(* CODESYS project sensata_io.library
   Company: Sensata Technologies
   DocFormat: reStructuredText
   Description: Contains IO structs for easy linking to IO
   Version: 0.0.1
   Placeholder: Sensata_IO
   Title: Sensata_IO

Project tree, tasks and I/O mapping:
  libraries: Tc2_Standard, * (Beckhoff Automation GmbH); Tc2_System, * (Beckhoff Automation GmbH); Tc2_Utilities, * (Beckhoff Automation GmbH); Tc3_Module, * (Beckhoff Automation GmbH)
  Beckhoff/
    EL1xxx/
      data type ST_EL1008
      data type ST_EL1008_Inputs
      data type ST_EL1014
      data type ST_EL1014_Inputs
      data type ST_EL1258
      data type ST_EL1258_Inputs
      data type ST_EL1258_Inputs_Channel
      data type ST_EL1258_Inputs_Channel_EventStates
      data type ST_EL1258_Inputs_Channel_Status
      data type ST_EL1258_Outputs
      data type ST_EL1258_Outputs_Channel
    EL2xxx/
      data type ST_EL2004
      data type ST_EL2004_Outputs
      data type ST_EL2008
      data type ST_EL2008_Outputs
      data type ST_EL2624
      data type ST_EL2624_Outputs
    EL3xxx/
      data type ST_EL3104
      data type ST_EL3104_Inputs
      data type ST_EL3104_Inputs_Channel
      data type ST_EL3104_Inputs_Channel_Status
      data type ST_EL3704_24BitVoltageDiff
      data type ST_EL3704_24BitVoltageDiff_Inputs
      data type ST_EL3704_24BitVoltageDiff_Inputs_Status
      data type ST_EL3773
      data type ST_EL3773_Inputs
      data type ST_EL3773_Inputs_Channel
      data type ST_EL3773_Inputs_Channel_Status
    EP1xxx/
      data type ST_EP1008
      data type ST_EP1008_Inputs
  IO Debug/
    function F_LinkDigitalIOStructs [ST]
    function F_SetDigitalInput [ST]
    function F_SetDigitalOutput [ST]
    data type ST_DebugDigitalIO
  Keyence/
    Barcode Scanners/
      data type ST_KeyenceNL20_EIP
      data type ST_KeyenceNL20_EIP_Inputs
      data type ST_KeyenceNL20_EIP_Outputs
      data type ST_KeyenceSR750_EIP
      data type ST_KeyenceSR750_EIP_Inputs
      data type ST_KeyenceSR750_EIP_Outputs
      data type ST_KeyenceSRX1H3H_EIP
      data type ST_KeyenceSRX1H3H_EIP_Inputs
      data type ST_KeyenceSRX1H3H_EIP_Outputs
    Height Check/
      data type ST_DLEC1A
      data type ST_DLEC1A_Inputs
      data type ST_DLEC1A_Inputs_Response
      data type ST_DLEC1A_Inputs_SystemStatus
      data type ST_DLEC1A_Outputs
      data type ST_DLEC1A_Outputs_Request
    Safety PLCs/
    Sensors/
      data type ST_LRX100
      data type ST_LRX100_Inputs
      data type ST_LRX100_Outputs
  MurrElektronik/
    data type ST_IMPACT67
    data type ST_IMPACT67_Inputs
  Norgren/
    data type ST_VR10
    data type ST_VR10_Inputs
    data type ST_VR10_Outputs
  SMC/
    data type ST_SMCEX260SEC3
    data type ST_SMCEX260SEC3_32Bit
    data type ST_SMCEX260SEC3_32Bit_Outputs
    data type ST_SMCEX260SEC3_Outputs
*)

// Beckhoff/EL1xxx/ST_EL1008
TYPE ST_EL1008 :
STRUCT
	stIn AT %I*: ST_EL1008_Inputs;
END_STRUCT
END_TYPE

// Beckhoff/EL1xxx/ST_EL1008_Inputs
TYPE ST_EL1008_Inputs :
STRUCT
	bitInput1: BIT;
	bitInput2: BIT;
	bitInput3: BIT;
	bitInput4: BIT;
	bitInput5: BIT;
	bitInput6: BIT;
	bitInput7: BIT;
	bitInput8: BIT;
END_STRUCT
END_TYPE

// Beckhoff/EL1xxx/ST_EL1014
TYPE ST_EL1014 :
STRUCT
	stIn AT %I*: ST_EL1014_Inputs;
END_STRUCT
END_TYPE

// Beckhoff/EL1xxx/ST_EL1014_Inputs
TYPE ST_EL1014_Inputs :
STRUCT
	bitInput1: BIT;
	bitInput2: BIT;
	bitInput3: BIT;
	bitInput4: BIT;
END_STRUCT
END_TYPE

// Beckhoff/EL1xxx/ST_EL1258
TYPE ST_EL1258 :
STRUCT
	stIn AT %I*: ST_EL1258_Inputs;
	stOut AT %Q*: ST_EL1258_Outputs;
END_STRUCT
END_TYPE

// Beckhoff/EL1xxx/ST_EL1258_Inputs
TYPE ST_EL1258_Inputs :
STRUCT
	stChannel1: ST_EL1258_Inputs_Channel;
	stChannel2: ST_EL1258_Inputs_Channel;
	stChannel3: ST_EL1258_Inputs_Channel;
	stChannel4: ST_EL1258_Inputs_Channel;
	stChannel5: ST_EL1258_Inputs_Channel;
	stChannel6: ST_EL1258_Inputs_Channel;
	stChannel7: ST_EL1258_Inputs_Channel;
	stChannel8: ST_EL1258_Inputs_Channel;
END_STRUCT
END_TYPE

// Beckhoff/EL1xxx/ST_EL1258_Inputs_Channel
TYPE ST_EL1258_Inputs_Channel :
STRUCT
	stStatus: ST_EL1258_Inputs_Channel_Status;
	stEventStates: ST_EL1258_Inputs_Channel_EventStates;
	arrEventTime: ARRAY[1..10] OF UDINT;
END_STRUCT
END_TYPE

// Beckhoff/EL1xxx/ST_EL1258_Inputs_Channel_EventStates
TYPE ST_EL1258_Inputs_Channel_EventStates :
STRUCT
	bitEventState01: BIT;
	bitEventState02: BIT;
	bitEventState03: BIT;
	bitEventState04: BIT;
	bitEventState05: BIT;
	bitEventState06: BIT;
	bitEventState07: BIT;
	bitEventState08: BIT;
	bitEventState09: BIT;
	bitEventState10: BIT;
END_STRUCT
END_TYPE

// Beckhoff/EL1xxx/ST_EL1258_Inputs_Channel_Status
TYPE ST_EL1258_Inputs_Channel_Status :
STRUCT
	usintEventsCount: USINT;
	
	bitState: BIT;
	bitBufferOverflow: BIT;
	{attribute 'hide'}
	bitReserved022: BIT;
	{attribute 'hide'}
	bitReserved023: BIT;
	{attribute 'hide'}
	bitReserved024: BIT;
	{attribute 'hide'}
	bitReserved25: BIT;
	bitCycleCountBit0: BIT;
	bitCycleCountBit1: BIT;
	
	usintBufferEvents: USINT;
	usintOrderFeedback: USINT;
END_STRUCT
END_TYPE

// Beckhoff/EL1xxx/ST_EL1258_Outputs
TYPE ST_EL1258_Outputs :
STRUCT
	stChannel1: ST_EL1258_Outputs_Channel;
	stChannel2: ST_EL1258_Outputs_Channel;
	stChannel3: ST_EL1258_Outputs_Channel;
	stChannel4: ST_EL1258_Outputs_Channel;
	stChannel5: ST_EL1258_Outputs_Channel;
	stChannel6: ST_EL1258_Outputs_Channel;
	stChannel7: ST_EL1258_Outputs_Channel;
	stChannel8: ST_EL1258_Outputs_Channel;
END_STRUCT
END_TYPE

// Beckhoff/EL1xxx/ST_EL1258_Outputs_Channel
TYPE ST_EL1258_Outputs_Channel :
STRUCT
	bitBufferReset: BIT;
	{attribute 'hide'}
	bitReserved01: BIT;
	{attribute 'hide'}
	bitReserved02: BIT;
	{attribute 'hide'}
	bitReserved03: BIT;
	{attribute 'hide'}
	bitReserved04: BIT;
	{attribute 'hide'}
	bitReserved05: BIT;
	{attribute 'hide'}
	bitReserved06: BIT;
	{attribute 'hide'}
	bitReserved07: BIT;
	
	{attribute 'hide'}
	byteReserved10: BYTE;
	
	usintInputOrderCounter: BOOL;
END_STRUCT
END_TYPE

// Beckhoff/EL2xxx/ST_EL2004
TYPE ST_EL2004 :
STRUCT
	stOut AT %Q*: ST_EL2004_Outputs;
END_STRUCT
END_TYPE

// Beckhoff/EL2xxx/ST_EL2004_Outputs
TYPE ST_EL2004_Outputs :
STRUCT
	bitOutput1: BIT;
	bitOutput2: BIT;
	bitOutput3: BIT;
	bitOutput4: BIT;
END_STRUCT
END_TYPE

// Beckhoff/EL2xxx/ST_EL2008
TYPE ST_EL2008 :
STRUCT
	stOut AT %Q*: ST_EL2008_Outputs;
END_STRUCT
END_TYPE

// Beckhoff/EL2xxx/ST_EL2008_Outputs
TYPE ST_EL2008_Outputs :
STRUCT
	bitOutput1: BIT;
	bitOutput2: BIT;
	bitOutput3: BIT;
	bitOutput4: BIT;
	bitOutput5: BIT;
	bitOutput6: BIT;
	bitOutput7: BIT;
	bitOutput8: BIT;
END_STRUCT
END_TYPE

// Beckhoff/EL2xxx/ST_EL2624
TYPE ST_EL2624 :
STRUCT
	stOut AT %Q*: ST_EL2624_Outputs;
END_STRUCT
END_TYPE

// Beckhoff/EL2xxx/ST_EL2624_Outputs
TYPE ST_EL2624_Outputs :
STRUCT
	bitRelay1: BIT;
	bitRelay2: BIT;
	bitRelay3: BIT;
	bitRelay4: BIT;
END_STRUCT
END_TYPE

// Beckhoff/EL3xxx/ST_EL3104
TYPE ST_EL3104 :
STRUCT
	stIn AT %I*: ST_EL3104_Inputs;
END_STRUCT
END_TYPE

// Beckhoff/EL3xxx/ST_EL3104_Inputs
TYPE ST_EL3104_Inputs :
STRUCT
	stChannel1: ST_EL3104_Inputs_Channel;
	stChannel2: ST_EL3104_Inputs_Channel;
	stChannel3: ST_EL3104_Inputs_Channel;
	stChannel4: ST_EL3104_Inputs_Channel;
END_STRUCT
END_TYPE

// Beckhoff/EL3xxx/ST_EL3104_Inputs_Channel
TYPE ST_EL3104_Inputs_Channel :
STRUCT
	stStatus: ST_EL3104_Inputs_Channel_Status;
	intValue: INT;
END_STRUCT
END_TYPE

// Beckhoff/EL3xxx/ST_EL3104_Inputs_Channel_Status
TYPE ST_EL3104_Inputs_Channel_Status :
STRUCT
	bitUnderRange: BIT;
	bitOverRange: BIT;
	bitOverLimit1: BIT;
	bitUnderLimit1: BIT;
	bitOverLimit2: BIT;
	bitUnderLimit2: BIT;
	bitError: BIT;
	{attribute 'hide'}
	bitReserved07: BIT;
	
	{attribute 'hide'}
	bitReserved10: BIT;
	{attribute 'hide'}
	bitReserved11: BIT;
	{attribute 'hide'}
	bitReserved12: BIT;
	{attribute 'hide'}
	bitReserved13: BIT;
	{attribute 'hide'}
	bitReserved14: BIT;
	bitSyncError: BIT;
	bitTxPDOState: BIT;
	bitTxPDOToggle: BIT;
END_STRUCT
END_TYPE

// Beckhoff/EL3xxx/ST_EL3704_24BitVoltageDiff
TYPE ST_EL3704_24BitVoltageDiff :
STRUCT
	stIn AT %I*: ST_EL3704_24BitVoltageDiff_Inputs;
END_STRUCT
END_TYPE

// Beckhoff/EL3xxx/ST_EL3704_24BitVoltageDiff_Inputs
TYPE ST_EL3704_24BitVoltageDiff_Inputs :
STRUCT
	stChannel1Status: ST_EL3704_24BitVoltageDiff_Inputs_Status;
	dintChannel1Value: DINT;
	ulintChannel1Timestamp: ULINT;
	stChannel2Status: ST_EL3704_24BitVoltageDiff_Inputs_Status;
	dintChannel2Value: DINT;
	stChannel3Status: ST_EL3704_24BitVoltageDiff_Inputs_Status;
	dintChannel3Value: DINT;
	stChannel4Status: ST_EL3704_24BitVoltageDiff_Inputs_Status;
	dintChannel4Value: DINT;
END_STRUCT
END_TYPE

// Beckhoff/EL3xxx/ST_EL3704_24BitVoltageDiff_Inputs_Status
TYPE ST_EL3704_24BitVoltageDiff_Inputs_Status :
STRUCT
	usintSamples: USINT;
	bitError: BIT;
	bitUnderrange: BIT;
	bitOverrange: BIT;
	{attribute 'hide'}
	bitReserved13: BIT;
	bitDiag: BIT;
	bitTxPDOState: BIT;
	bitCycleCount1: BIT;
	bitCycleCount2: BIT;
END_STRUCT
END_TYPE

// Beckhoff/EL3xxx/ST_EL3773
TYPE ST_EL3773 :
STRUCT
	stIn AT %I*: ST_EL3773_Inputs;
END_STRUCT
END_TYPE

// Beckhoff/EL3xxx/ST_EL3773_Inputs
TYPE ST_EL3773_Inputs :
STRUCT
	stL1: ST_EL3773_Inputs_Channel;
	stL2: ST_EL3773_Inputs_Channel;
	stL3: ST_EL3773_Inputs_Channel;
	udintNextSyncTimeLow: UDINT;
	udintNextSyncTimeHigh: UDINT;
	uintSampleCount: UINT;
END_STRUCT
END_TYPE

// Beckhoff/EL3xxx/ST_EL3773_Inputs_Channel
TYPE ST_EL3773_Inputs_Channel :
STRUCT
	stVoltageStatus: ST_EL3773_Inputs_Channel_Status;
	arrVoltageSamples: ARRAY[0..9] OF INT;
	stCurrentStatus: ST_EL3773_Inputs_Channel_Status;
	arrCurrentSamples: ARRAY[0..9] OF INT;
END_STRUCT
END_TYPE

// Beckhoff/EL3xxx/ST_EL3773_Inputs_Channel_Status
TYPE ST_EL3773_Inputs_Channel_Status :
STRUCT
	bitUnderRange: BIT;
	bitOverRange: BIT;
	bitOverLimit: BIT;
	bitUnderLimit: BIT;
	{attribute 'hide'}
	bitReserved04: BIT;
	{attribute 'hide'}
	bitReserved05: BIT;
	bitError: BIT;
	{attribute 'hide'}
	bitReserved07: BIT;
	
	{attribute 'hide'}
	bitReserved10: BIT;
	{attribute 'hide'}
	bitReserved11: BIT;
	{attribute 'hide'}
	bitReserved12: BIT;
	{attribute 'hide'}
	bitReserved13: BIT;
	{attribute 'hide'}
	bitReserved14: BIT;
	bitSyncError: BIT;
	bitTxPDOState: BIT;
	bitTxPDOToggle: BIT;
END_STRUCT
END_TYPE

// Beckhoff/EP1xxx/ST_EP1008
TYPE ST_EP1008 :
STRUCT
	stIn AT %I*: ST_EP1008_Inputs;
END_STRUCT
END_TYPE

// Beckhoff/EP1xxx/ST_EP1008_Inputs
TYPE ST_EP1008_Inputs :
STRUCT
	bitInput1: BIT;
	bitInput2: BIT;
	bitInput3: BIT;
	bitInput4: BIT;
	bitInput5: BIT;
	bitInput6: BIT;
	bitInput7: BIT;
	bitInput8: BIT;
END_STRUCT
END_TYPE

// IO Debug/ST_DebugDigitalIO
TYPE ST_DebugDigitalIO :
STRUCT
	(* Label for this IO. *)
	strLabel: T_MaxString;
	(* Current value. *)
	bCurrentValue: BOOL;
	(* Set to TRUE if IO is an output. *)
	bOutput: BOOL;
	(* Set TRUE to force output to a value. *)
	bForce: BOOL;
	(* Value to force output to. *)
	bForceValue: BOOL;
END_STRUCT
END_TYPE

// Keyence/Barcode Scanners/ST_KeyenceNL20_EIP
TYPE ST_KeyenceNL20_EIP :
STRUCT
	stIn AT %I*: ST_KeyenceNL20_EIP_Inputs;
	stOut AT %Q*: ST_KeyenceNL20_EIP_Outputs;
END_STRUCT
END_TYPE

// Keyence/Barcode Scanners/ST_KeyenceNL20_EIP_Inputs
TYPE ST_KeyenceNL20_EIP_Inputs :
STRUCT
	bitError: BIT;
	bitResponseDataAvailable: BIT;
	bitResultDataStrobe: BIT;
	{attribute 'hide'}
	bitReserved003: BIT;
	{attribute 'hide'}
	bitReserved004: BIT;
	{attribute 'hide'}
	bitReserved005: BIT;
	bitBufferOverflowError: BIT;
	bitGeneralError: BIT;
	
	bitBusy: BIT;
	{attribute 'hide'}
	bitReserved011: BIT;
	{attribute 'hide'}
	bitReserved012: BIT;
	bitModeBusy: BIT;
	{attribute 'hide'}
	bitReserved014: BIT;
	{attribute 'hide'}
	bitReserved015: BIT;
	{attribute 'hide'}
	bitReserved016: BIT;
	{attribute 'hide'}
	bitReserved017: BIT;
	
	bitReadComplete: BIT;
	{attribute 'hide'}
	bitReserved021: BIT;
	{attribute 'hide'}
	bitReserved022: BIT;
	{attribute 'hide'}
	bitReserved023: BIT;
	{attribute 'hide'}
	bitReserved024: BIT;
	{attribute 'hide'}
	bitReserved025: BIT;
	{attribute 'hide'}
	bitReserved026: BIT;
	{attribute 'hide'}
	bitReserved027: BIT;
	
	{attribute 'hide'}
	byteReserved030: BYTE;

	bitIN1Status: BIT;
	bitIN2Status: BIT;
	{attribute 'hide'}
	bitReserved042: BIT;
	{attribute 'hide'}
	bitReserved043: BIT;
	bitOUT1Status: BIT;
	bitOUT2Status: BIT;
	bitOUT3Status: BIT;
	bitOUT4Status: BIT;
	
	{attribute 'hide'}
	arrReserved050: ARRAY[0..26] OF BYTE;
	
	uintGeneralErrorCode: UINT;
	
	{attribute 'hide'}
	wordReserved340: WORD;
	
	uintResultDataReadyCount: UINT;
	uintResultDataUpdateCount: UINT;
	
	{attribute 'hide'}
	wordReserved400: WORD;
	
	uintResultDataSize: UINT;
	arrResultData: ARRAY[0..127] OF BYTE;
END_STRUCT
END_TYPE

// Keyence/Barcode Scanners/ST_KeyenceNL20_EIP_Outputs
TYPE ST_KeyenceNL20_EIP_Outputs :
STRUCT
	{attribute 'hide'}
	bitReserved000: BIT;
	bitResultDataLatch: BIT;
	{attribute 'hide'}
	bitReserved002: BIT;
	{attribute 'hide'}
	bitReserved003: BIT;
	{attribute 'hide'}
	bitReserved004: BIT;
	{attribute 'hide'}
	bitReserved005: BIT;
	{attribute 'hide'}
	bitReserved006: BIT;
	bitErrorClear: BIT;
	
	bitReadRequest: BIT;
	{attribute 'hide'}
	bitReserved011: BIT;
	{attribute 'hide'}
	bitReserved012: BIT;
	{attribute 'hide'}
	bitReserved013: BIT;
	{attribute 'hide'}
	bitReserved014: BIT;
	{attribute 'hide'}
	bitReserved015: BIT;
	{attribute 'hide'}
	bitReserved016: BIT;
	{attribute 'hide'}
	bitReserved017: BIT;
	
	bitReadCompleteClear: BIT;
	{attribute 'hide'}
	bitReserved021: BIT;
	{attribute 'hide'}
	bitReserved022: BIT;
	{attribute 'hide'}
	bitReserved023: BIT;
	{attribute 'hide'}
	bitReserved024: BIT;
	{attribute 'hide'}
	bitReserved025: BIT;
	{attribute 'hide'}
	bitReserved026: BIT;
	{attribute 'hide'}
	bitReserved027: BIT;
	
	{attribute 'hide'}
	byteReserved030: BYTE;
	
	uintBankNumber: UINT;
	
	{attribute 'hide'}
	arrReserved060: ARRAY[0..69] OF BYTE;
END_STRUCT
END_TYPE

// Keyence/Barcode Scanners/ST_KeyenceSR750_EIP
TYPE ST_KeyenceSR750_EIP :
STRUCT
	stIn AT %I*: ST_KeyenceSR750_EIP_Inputs;
	stOut AT %Q*: ST_KeyenceSR750_EIP_Outputs;
END_STRUCT
END_TYPE

// Keyence/Barcode Scanners/ST_KeyenceSR750_EIP_Inputs
TYPE ST_KeyenceSR750_EIP_Inputs :
STRUCT
	bitError: BIT;
	bitResponseDataAvailable: BIT;
	bitResultDataStrobe: BIT;
	{attribute 'hide'}
	bitReserved003: BIT;
	{attribute 'hide'}
	bitReserved004: BIT;
	{attribute 'hide'}
	bitReserved005: BIT;
	bitBufferOverflowError: BIT;
	bitGeneralError: BIT;
	
	bitBusy: BIT;
	bitTrgBusy: BIT;
	bitLockBusy: BIT;
	bitModeBusy: BIT;
	bitErrBusy: BIT;
	{attribute 'hide'}
	bitReserved015: BIT;
	{attribute 'hide'}
	bitReserved016: BIT;
	{attribute 'hide'}
	bitReserved017: BIT;
	
	bitReadComplete: BIT;
	bitPresetComplete: BIT;
	bitRegisterPresetDataComplete: BIT;
	bitTuneComplete: BIT;
	{attribute 'hide'}
	bitReserved024: BIT;
	{attribute 'hide'}
	bitReserved025: BIT;
	{attribute 'hide'}
	bitReserved026: BIT;
	bitExtRequestComplete: BIT;
	
	bitReadFailure: BIT;
	bitPresetFailure: BIT;
	bitRegisterPresetDataFailure: BIT;
	bitTuneFailure: BIT;
	{attribute 'hide'}
	bitReserved034: BIT;
	{attribute 'hide'}
	bitReserved035: BIT;
	{attribute 'hide'}
	bitReserved036: BIT;
	bitExtRequestFailure: BIT;

	bitIN1Status: BIT;
	bitIN2Status: BIT;
	{attribute 'hide'}
	bitReserved042: BIT;
	{attribute 'hide'}
	bitReserved043: BIT;
	bitOUT1Status: BIT;
	bitOUT2Status: BIT;
	bitOUT3Status: BIT;
	{attribute 'hide'}
	bitReserved047: BIT;
	
	bitUnstable: BIT;
	bitMatchingLevelUnstable: BIT;
	bitISOIEC15415Unstable: BIT;
	bitAIMDPMUnstable: BIT;
	bitSAEAS9132Unstable: BIT;
	{attribute 'hide'}
	bitReserved055: BIT;
	{attribute 'hide'}
	bitReserved056: BIT;
	{attribute 'hide'}
	bitReserved057: BIT;
	
	{attribute 'hide'}
	wordReserved060: WORD;
	
	uintMatchingLevel: UINT;
	uintISOIEC15415Grade: UINT;
	uintAIMDPMGrade: UINT;
	
	{attribute 'hide'}
	wordReserved140: WORD;
	
	uintReadResultCode: UINT;
	uintPresetResultCode: UINT;
	uintRegisterPresetDataResultCode: UINT;
	uintTuningResultCode: UINT;
	
	{attribute 'hide'}
	arrReserved240: ARRAY[0..2] OF WORD;
	
	uintExtRequestResultCode: UINT;
	uintGeneralErrorCode: UINT;
	
	{attribute 'hide'}
	wordReserved340: WORD;
	
	uintResultDataReadyCount: UINT;
	uintResultDataUpdateCount: UINT;
	
	{attribute 'hide'}
	wordReserved400: WORD;
	
	uintResultDataSize: UINT;
	arrResultData: ARRAY[0..127] OF BYTE;
END_STRUCT
END_TYPE

// Keyence/Barcode Scanners/ST_KeyenceSR750_EIP_Outputs
TYPE ST_KeyenceSR750_EIP_Outputs :
STRUCT
	{attribute 'hide'}
	bitReserved000: BIT;
	bitResultDataLatch: BIT;
	{attribute 'hide'}
	bitReserved002: BIT;
	{attribute 'hide'}
	bitReserved003: BIT;
	{attribute 'hide'}
	bitReserved004: BIT;
	{attribute 'hide'}
	bitReserved005: BIT;
	{attribute 'hide'}
	bitReserved006: BIT;
	bitErrorClear: BIT;
	
	bitReadRequest: BIT;
	bitPresetRequest: BIT;
	bitRegisterPresetDataRequest: BIT;
	bitTuneRequest: BIT;
	{attribute 'hide'}
	bitReserved014: BIT;
	{attribute 'hide'}
	bitReserved015: BIT;
	{attribute 'hide'}
	bitReserved016: BIT;
	{attribute 'hide'}
	bitReserved017: BIT;
	
	bitReadCompleteClear: BIT;
	bitPresetCompleteClear: BIT;
	bitRegisterPresetDataCompleteClear: BIT;
	bitTuneCompleteClear: BIT;
	{attribute 'hide'}
	bitReserved024: BIT;
	{attribute 'hide'}
	bitReserved025: BIT;
	{attribute 'hide'}
	bitReserved026: BIT;
	bitExtRequestCompleteClear: BIT;
	
	{attribute 'hide'}
	byteReserved030: BYTE;
	
	uintBankNumber: UINT;
	
	{attribute 'hide'}
	arrReserved060: ARRAY[0..1] OF WORD;
	
	uintUserDataSize: UINT;
	arrUserData: ARRAY[0..63] OF BYTE;
END_STRUCT
END_TYPE

// Keyence/Barcode Scanners/ST_KeyenceSRX1H3H_EIP
TYPE ST_KeyenceSRX1H3H_EIP :
STRUCT
	stIn AT %I*: ST_KeyenceSRX1H3H_EIP_Inputs;
	stOut AT %Q*: ST_KeyenceSRX1H3H_EIP_Outputs;
END_STRUCT
END_TYPE

// Keyence/Barcode Scanners/ST_KeyenceSRX1H3H_EIP_Inputs
TYPE ST_KeyenceSRX1H3H_EIP_Inputs :
STRUCT
	bitError: BIT;
	bitResponseDataAvailable: BIT;
	bitResultDataStrobe: BIT;
	{attribute 'hide'}
	bitReserved003: BIT;
	{attribute 'hide'}
	bitReserved004: BIT;
	{attribute 'hide'}
	bitReserved005: BIT;
	bitBufferOverflowError: BIT;
	bitGeneralError: BIT;
	
	bitBusy: BIT;
	bitTrgBusy: BIT;
	bitLockBusy: BIT;
	bitModeBusy: BIT;
	bitErrBusy: BIT;
	{attribute 'hide'}
	bitReserved015: BIT;
	bitReady: BIT;
	{attribute 'hide'}
	bitReserved017: BIT;
	
	bitReadComplete: BIT;
	bitPresetComplete: BIT;
	bitRegisterPresetDataComplete: BIT;
	bitTuneComplete: BIT;
	bitBloadComplete: BIT;
	{attribute 'hide'}
	bitReserved025: BIT;
	{attribute 'hide'}
	bitReserved026: BIT;
	bitExtRequestComplete: BIT;
	
	bitReadFailure: BIT;
	bitPresetFailure: BIT;
	bitRegisterPresetDataFailure: BIT;
	bitTuneFailure: BIT;
	bitBloadFailure: BIT;
	{attribute 'hide'}
	bitReserved035: BIT;
	{attribute 'hide'}
	bitReserved036: BIT;
	bitExtRequestFailure: BIT;

	bitIN1Status: BIT;
	bitIN2Status: BIT;
	{attribute 'hide'}
	bitReserved042: BIT;
	{attribute 'hide'}
	bitReserved043: BIT;
	bitOUT1Status: BIT;
	bitOUT2Status: BIT;
	bitOUT3Status: BIT;
	{attribute 'hide'}
	bitReserved047: BIT;
	
	bitUnstable: BIT;
	bitMatchingLevelUnstable: BIT;
	bitISOIEC15415Unstable: BIT;
	bitAIMDPMUnstable: BIT;
	bitSAEAS9132Unstable: BIT;
	{attribute 'hide'}
	bitReserved055: BIT;
	{attribute 'hide'}
	bitReserved056: BIT;
	{attribute 'hide'}
	bitReserved057: BIT;
	
	{attribute 'hide'}
	wordReserved060: WORD;
	
	uintMatchingLevel: UINT;
	uintISOIEC15415Grade: UINT;
	uintAIMDPMGrade: UINT;
	
	{attribute 'hide'}
	wordReserved140: WORD;
	
	uintReadResultCode: UINT;
	uintPresetResultCode: UINT;
	uintRegisterPresetDataResultCode: UINT;
	uintTuningResultCode: UINT;
	
	{attribute 'hide'}
	arrReserved240: ARRAY[0..2] OF WORD;
	
	uintExtRequestResultCode: UINT;
	uintGeneralErrorCode: UINT;
	
	{attribute 'hide'}
	wordReserved340: WORD;
	
	uintResultDataReadyCount: UINT;
	uintResultDataUpdateCount: UINT;
	
	{attribute 'hide'}
	wordReserved400: WORD;
	
	uintResultDataSize: UINT;
	arrResultData: ARRAY[0..127] OF BYTE;
END_STRUCT
END_TYPE

// Keyence/Barcode Scanners/ST_KeyenceSRX1H3H_EIP_Outputs
TYPE ST_KeyenceSRX1H3H_EIP_Outputs :
STRUCT
	{attribute 'hide'}
	bitReserved000: BIT;
	bitResultDataLatch: BIT;
	{attribute 'hide'}
	bitReserved002: BIT;
	{attribute 'hide'}
	bitReserved003: BIT;
	{attribute 'hide'}
	bitReserved004: BIT;
	{attribute 'hide'}
	bitReserved005: BIT;
	{attribute 'hide'}
	bitReserved006: BIT;
	bitErrorClear: BIT;
	
	bitReadRequest: BIT;
	bitPresetRequest: BIT;
	bitRegisterPresetDataRequest: BIT;
	bitTuneRequest: BIT;
	{attribute 'hide'}
	bitReserved014: BIT;
	{attribute 'hide'}
	bitReserved015: BIT;
	{attribute 'hide'}
	bitReserved016: BIT;
	{attribute 'hide'}
	bitReserved017: BIT;
	
	bitReadCompleteClear: BIT;
	bitPresetCompleteClear: BIT;
	bitRegisterPresetDataCompleteClear: BIT;
	bitTuneCompleteClear: BIT;
	{attribute 'hide'}
	bitReserved024: BIT;
	{attribute 'hide'}
	bitReserved025: BIT;
	{attribute 'hide'}
	bitReserved026: BIT;
	bitExtRequestCompleteClear: BIT;
	
	{attribute 'hide'}
	byteReserved030: BYTE;
	
	uintBankNumber: UINT;
	
	{attribute 'hide'}
	arrReserved060: ARRAY[0..1] OF WORD;
	
	uintUserDataSize: UINT;
	arrUserData: ARRAY[0..63] OF BYTE;
END_STRUCT
END_TYPE

// Keyence/Height Check/ST_DLEC1A
TYPE ST_DLEC1A :
STRUCT
	stIn AT %I*: ST_DLEC1A_Inputs;
	stOut AT %Q*: ST_DLEC1A_Outputs;
END_STRUCT
END_TYPE

// Keyence/Height Check/ST_DLEC1A_Inputs
TYPE ST_DLEC1A_Inputs :
STRUCT
	stSystemStatus: ST_DLEC1A_Inputs_SystemStatus;
	{attribute 'hide'}
	arrUnused: ARRAY[1..5] OF DWORD;
	arrCurrentValue: ARRAY[1..8] OF DINT;
	stResponse: ST_DLEC1A_Inputs_Response;
END_STRUCT
END_TYPE

// Keyence/Height Check/ST_DLEC1A_Inputs_Response
TYPE ST_DLEC1A_Inputs_Response :
STRUCT
	bitMainProgChgAck: BIT;
	bitMainTriggerAck: BIT;
	bitMainZeroOffsetAck: BIT;
	bitMainValueUpdateAck: BIT;
	bitMainEmissionStopAck: BIT;
	{attribute 'hide'}
	bitReserved005: BIT;
	{attribute 'hide'}
	bitReserved006: BIT;
	{attribute 'hide'}
	bitReserved007: BIT;
	
	{attribute 'hide'}
	bitReserved010: BIT;
	bitValue1Invalid: BIT;
	bitValue1UnderRange: BIT;
	bitValue1OverRange: BIT;
	{attribute 'hide'}
	bitReserved014: BIT;
	{attribute 'hide'}
	bitReserved015: BIT;
	bitMainWarning: BIT;
	bitMainError: BIT;
	
	bitMainOutput01: BIT;
	bitMainOutput02: BIT;
	bitMainOutput03: BIT;
	bitMainOutput04: BIT;
	bitMainOutput05: BIT;
	{attribute 'hide'}
	bitReserved025: BIT;
	{attribute 'hide'}
	bitReserved026: BIT;
	{attribute 'hide'}
	bitReserved027: BIT;
	
	{attribute 'hide'}
	bitReserved030: BIT;
	bitValue2Invalid: BIT;
	bitValue2UnderRange: BIT;
	bitValue2OverRange: BIT;
	{attribute 'hide'}
	bitReserved034: BIT;
	{attribute 'hide'}
	bitReserved035: BIT;
	{attribute 'hide'}
	bitReserved036: BIT;
	{attribute 'hide'}
	bitReserved037: BIT;
	
	bitMainOutput06: BIT;
	bitMainOutput07: BIT;
	bitMainOutput08: BIT;
	bitMainOutput09: BIT;
	bitMainOutput10: BIT;
	{attribute 'hide'}
	bitReserved045: BIT;
	{attribute 'hide'}
	bitReserved046: BIT;
	{attribute 'hide'}
	bitReserved047: BIT;
	
	{attribute 'hide'}
	bitReserved050: BIT;
	bitValue3Invalid: BIT;
	bitValue3UnderRange: BIT;
	bitValue3OverRange: BIT;
	{attribute 'hide'}
	bitReserved054: BIT;
	{attribute 'hide'}
	bitReserved055: BIT;
	{attribute 'hide'}
	bitReserved056: BIT;
	{attribute 'hide'}
	bitReserved057: BIT;
	
	bitExpProgChgAck: BIT;
	bitExpTriggerAck: BIT;
	bitExpZeroOffsetAck: BIT;
	bitExpValueUpdateAck: BIT;
	bitExpEmissionStopAck: BIT;
	{attribute 'hide'}
	bitReserved065: BIT;
	{attribute 'hide'}
	bitReserved066: BIT;
	{attribute 'hide'}
	bitReserved067: BIT;
	
	{attribute 'hide'}
	bitReserved070: BIT;
	bitValue4Invalid: BIT;
	bitValue4UnderRange: BIT;
	bitValue4OverRange: BIT;
	{attribute 'hide'}
	bitReserved074: BIT;
	{attribute 'hide'}
	bitReserved075: BIT;
	bitExpWarning: BIT;
	bitExpError: BIT;
	
	bitExpOutput01: BIT;
	bitExpOutput02: BIT;
	bitExpOutput03: BIT;
	bitExpOutput04: BIT;
	bitExpOutput05: BIT;
	{attribute 'hide'}
	bitReserved085: BIT;
	{attribute 'hide'}
	bitReserved086: BIT;
	{attribute 'hide'}
	bitReserved087: BIT;
	
	{attribute 'hide'}
	bitReserved090: BIT;
	bitValue5Invalid: BIT;
	bitValue5UnderRange: BIT;
	bitValue5OverRange: BIT;
	{attribute 'hide'}
	bitReserved094: BIT;
	{attribute 'hide'}
	bitReserved095: BIT;
	{attribute 'hide'}
	bitReserved096: BIT;
	{attribute 'hide'}
	bitReserved097: BIT;
	
	bitExpOutput06: BIT;
	bitExpOutput07: BIT;
	bitExpOutput08: BIT;
	bitExpOutput09: BIT;
	bitExpOutput10: BIT;
	{attribute 'hide'}
	bitReserved105: BIT;
	{attribute 'hide'}
	bitReserved106: BIT;
	{attribute 'hide'}
	bitReserved107: BIT;
	
	{attribute 'hide'}
	bitReserved110: BIT;
	bitValue6Invalid: BIT;
	bitValue6UnderRange: BIT;
	bitValue6OverRange: BIT;
	{attribute 'hide'}
	bitReserved114: BIT;
	{attribute 'hide'}
	bitReserved115: BIT;
	{attribute 'hide'}
	bitReserved116: BIT;
	{attribute 'hide'}
	bitReserved117: BIT;
	
	{attribute 'hide'}
	byteReserved120: BYTE;
	
	{attribute 'hide'}
	bitReserved130: BIT;
	bitValue7Invalid: BIT;
	bitValue7UnderRange: BIT;
	bitValue7OverRange: BIT;
	{attribute 'hide'}
	bitReserved134: BIT;
	{attribute 'hide'}
	bitReserved135: BIT;
	{attribute 'hide'}
	bitReserved136: BIT;
	{attribute 'hide'}
	bitReserved137: BIT;
	
	{attribute 'hide'}
	byteReserved140: BYTE;
	
	{attribute 'hide'}
	bitReserved150: BIT;
	bitValue8Invalid: BIT;
	bitValue8UnderRange: BIT;
	bitValue8OverRange: BIT;
	{attribute 'hide'}
	bitReserved154: BIT;
	{attribute 'hide'}
	bitReserved155: BIT;
	{attribute 'hide'}
	bitReserved156: BIT;
	{attribute 'hide'}
	bitReserved157: BIT;
END_STRUCT
END_TYPE

// Keyence/Height Check/ST_DLEC1A_Inputs_SystemStatus
TYPE ST_DLEC1A_Inputs_SystemStatus :
STRUCT
	bitErrorStatus: BIT;
	bitWarningStatus: BIT;
	{attribute 'hide'}
	bitReserved02: BIT;
	bitCurrentValueProp: BIT;
	{attribute 'hide'}
	bitReserved04: BIT;
	{attribute 'hide'}
	bitReserved05: BIT;
	{attribute 'hide'}
	bitReserved06: BIT;
	{attribute 'hide'}
	bitReserved07: BIT;
	
	byteReserved10: BYTE;
	
	uintErrorCode: UINT;
END_STRUCT
END_TYPE

// Keyence/Height Check/ST_DLEC1A_Outputs
TYPE ST_DLEC1A_Outputs :
STRUCT
	stRequest: ST_DLEC1A_Outputs_Request;
END_STRUCT
END_TYPE

// Keyence/Height Check/ST_DLEC1A_Outputs_Request
TYPE ST_DLEC1A_Outputs_Request :
STRUCT
	{attribute 'hide'}
	bitReserved000: BIT;
	bitMainTrigger: BIT;
	bitMainProgChange: BIT;
	{attribute 'hide'}
	bitReserved003: BIT;
	bitExpTrigger: BIT;
	bitExpProgChange: BIT;
	{attribute 'hide'}
	bitReserved006: BIT;
	{attribute 'hide'}
	bitReserved007: BIT;
	
	{attribute 'hide'}
	byteReserved010: BYTE;
	{attribute 'hide'}
	wordReserved020: WORD;
	
	{attribute 'hide'}
	bitReserved040: BIT;
	bitMainZeroOffset: BIT;
	bitMainProgNumBit0: BIT;
	{attribute 'hide'}
	bitReserved043: BIT;
	bitExpZeroOffset: BIT;
	bitExpProgNumBit0: BIT;
	{attribute 'hide'}
	bitReserved046: BIT;
	{attribute 'hide'}
	bitReserved047: BIT;
	
	{attribute 'hide'}
	byteReserved050: BYTE;
	{attribute 'hide'}
	wordReserved060: WORD;
	
	{attribute 'hide'}
	bitReserved080: BIT;
	bitMainReset: BIT;
	bitMainProgNumBit1: BIT;
	{attribute 'hide'}
	bitReserved083: BIT;
	bitExpReset: BIT;
	bitExpProgNumBit1: BIT;
	{attribute 'hide'}
	bitReserved086: BIT;
	{attribute 'hide'}
	bitReserved087: BIT;
	
	{attribute 'hide'}
	byteReserved090: BYTE;
	{attribute 'hide'}
	wordReserved100: WORD;
	
	{attribute 'hide'}
	bitReserved120: BIT;
	bitMainEmissionStop: BIT;
	bitMainProgNumBit2: BIT;
	{attribute 'hide'}
	bitReserved123: BIT;
	bitExpEmissionStop: BIT;
	bitExpProgNumBit2: BIT;
	{attribute 'hide'}
	bitReserved126: BIT;
	{attribute 'hide'}
	bitReserved127: BIT;
	
	{attribute 'hide'}
	byteReserved130: BYTE;
	{attribute 'hide'}
	wordReserved140: WORD;
	
	{attribute 'hide'}
	bitReserved160: BIT;
	{attribute 'hide'}
	bitReserved161: BIT;
	bitMainProgNumBit3: BIT;
	{attribute 'hide'}
	bitReserved163: BIT;
	{attribute 'hide'}
	bitReserved164: BIT;
	bitExpProgNumBit3: BIT;
	{attribute 'hide'}
	bitReserved166: BIT;
	{attribute 'hide'}
	bitReserved167: BIT;
	
	{attribute 'hide'}
	byteReserved170: BYTE;
	{attribute 'hide'}
	wordReserved180: WORD;
END_STRUCT
END_TYPE

// Keyence/Sensors/ST_LRX100
TYPE ST_LRX100 :
STRUCT
	stIn AT %I*: ST_LRX100_Inputs;
	stOut AT %Q*: ST_LRX100_Outputs;
END_STRUCT
END_TYPE

// Keyence/Sensors/ST_LRX100_Inputs
TYPE ST_LRX100_Inputs :
STRUCT
	intValue: INT;
	{attribute 'hide'}
	bitReserved00: BIT;
	bitOvercurrent: BIT;
	bitHeadError: BIT;
	bitEEPROMError: BIT;
	{attribute 'hide'}
	bitReserved04: BIT;
	bitUserError: BIT;
	{attribute 'hide'}
	bitReserved06: BIT;
	{attribute 'hide'}
	bitReserved07: BIT;
	
	bitOutput1: BIT;
	bitOutput2: BIT;
	bitWarning: BIT;
	{attribute 'hide'}
	bitReserved13: BIT;
	{attribute 'hide'}
	bitReserved14: BIT;
	{attribute 'hide'}
	bitReserved15: BIT;
	{attribute 'hide'}
	bitReserved16: BIT;
	{attribute 'hide'}
	bitReserved17: BIT;
END_STRUCT
END_TYPE

// Keyence/Sensors/ST_LRX100_Outputs
TYPE ST_LRX100_Outputs :
STRUCT
	bInput: BIT;
END_STRUCT
END_TYPE

// MurrElektronik/ST_IMPACT67
TYPE ST_IMPACT67 :
STRUCT
	stIn AT %I*: ST_IMPACT67_Inputs;
END_STRUCT
END_TYPE

// MurrElektronik/ST_IMPACT67_Inputs
TYPE ST_IMPACT67_Inputs :
STRUCT
	bitInput00: BIT;
	bitInput01: BIT;
	bitInput02: BIT;
	bitInput03: BIT;
	bitInput04: BIT;
	bitInput05: BIT;
	bitInput06: BIT;
	bitInput07: BIT;
	
	bitInput10: BIT;
	bitInput11: BIT;
	bitInput12: BIT;
	bitInput13: BIT;
	bitInput14: BIT;
	bitInput15: BIT;
	bitInput16: BIT;
	bitInput17: BIT;
END_STRUCT
END_TYPE

// Norgren/ST_VR10
TYPE ST_VR10 :
STRUCT
	stIn AT %I*: ST_VR10_Inputs;
	stOut AT %Q*: ST_VR10_Outputs;
END_STRUCT
END_TYPE

// Norgren/ST_VR10_Inputs
TYPE ST_VR10_Inputs :
STRUCT
	usintModuleStatus: USINT;
	
	bitOutput00ShortCircuit: BIT;
	bitOutput01ShortCircuit: BIT;
	bitOutput02ShortCircuit: BIT;
	bitOutput03ShortCircuit: BIT;
	bitOutput04ShortCircuit: BIT;
	bitOutput05ShortCircuit: BIT;
	bitOutput06ShortCircuit: BIT;
	bitOutput07ShortCircuit: BIT;
	
	bitOutput10ShortCircuit: BIT;
	bitOutput11ShortCircuit: BIT;
	bitOutput12ShortCircuit: BIT;
	bitOutput13ShortCircuit: BIT;
	bitOutput14ShortCircuit: BIT;
	bitOutput15ShortCircuit: BIT;
	bitOutput16ShortCircuit: BIT;
	bitOutput17ShortCircuit: BIT;
	
	bitOutput20ShortCircuit: BIT;
	bitOutput21ShortCircuit: BIT;
	bitOutput22ShortCircuit: BIT;
	bitOutput23ShortCircuit: BIT;
	bitOutput24ShortCircuit: BIT;
	bitOutput25ShortCircuit: BIT;
	bitOutput26ShortCircuit: BIT;
	bitOutput27ShortCircuit: BIT;
	
	bitOutput00OpenLoad: BIT;
	bitOutput01OpenLoad: BIT;
	bitOutput02OpenLoad: BIT;
	bitOutput03OpenLoad: BIT;
	bitOutput04OpenLoad: BIT;
	bitOutput05OpenLoad: BIT;
	bitOutput06OpenLoad: BIT;
	bitOutput07OpenLoad: BIT;
	
	bitOutput10OpenLoad: BIT;
	bitOutput11OpenLoad: BIT;
	bitOutput12OpenLoad: BIT;
	bitOutput13OpenLoad: BIT;
	bitOutput14OpenLoad: BIT;
	bitOutput15OpenLoad: BIT;
	bitOutput16OpenLoad: BIT;
	bitOutput17OpenLoad: BIT;
	
	bitOutput20OpenLoad: BIT;
	bitOutput21OpenLoad: BIT;
	bitOutput22OpenLoad: BIT;
	bitOutput23OpenLoad: BIT;
	bitOutput24OpenLoad: BIT;
	bitOutput25OpenLoad: BIT;
	bitOutput26OpenLoad: BIT;
	bitOutput27OpenLoad: BIT;
	
	bitOutput00CycleOverrun: BIT;
	bitOutput01CycleOverrun: BIT;
	bitOutput02CycleOverrun: BIT;
	bitOutput03CycleOverrun: BIT;
	bitOutput04CycleOverrun: BIT;
	bitOutput05CycleOverrun: BIT;
	bitOutput06CycleOverrun: BIT;
	bitOutput07CycleOverrun: BIT;
	
	bitOutput10CycleOverrun: BIT;
	bitOutput11CycleOverrun: BIT;
	bitOutput12CycleOverrun: BIT;
	bitOutput13CycleOverrun: BIT;
	bitOutput14CycleOverrun: BIT;
	bitOutput15CycleOverrun: BIT;
	bitOutput16CycleOverrun: BIT;
	bitOutput17CycleOverrun: BIT;
	
	bitOutput20CycleOverrun: BIT;
	bitOutput21CycleOverrun: BIT;
	bitOutput22CycleOverrun: BIT;
	bitOutput23CycleOverrun: BIT;
	bitOutput24CycleOverrun: BIT;
	bitOutput25CycleOverrun: BIT;
	bitOutput26CycleOverrun: BIT;
	bitOutput27CycleOverrun: BIT;
END_STRUCT
END_TYPE

// Norgren/ST_VR10_Outputs
TYPE ST_VR10_Outputs :
STRUCT
	bitOutput00: BIT;
	bitOutput01: BIT;
	bitOutput02: BIT;
	bitOutput03: BIT;
	bitOutput04: BIT;
	bitOutput05: BIT;
	bitOutput06: BIT;
	bitOutput07: BIT;
	
	bitOutput10: BIT;
	bitOutput11: BIT;
	bitOutput12: BIT;
	bitOutput13: BIT;
	bitOutput14: BIT;
	bitOutput15: BIT;
	bitOutput16: BIT;
	bitOutput17: BIT;
	
	bitOutput20: BIT;
	bitOutput21: BIT;
	bitOutput22: BIT;
	bitOutput23: BIT;
	bitOutput24: BIT;
	bitOutput25: BIT;
	bitOutput26: BIT;
	bitOutput27: BIT;
END_STRUCT
END_TYPE

// SMC/ST_SMCEX260SEC3
TYPE ST_SMCEX260SEC3 :
STRUCT
	stOut AT %Q*: ST_SMCEX260SEC3_Outputs;
END_STRUCT
END_TYPE

// SMC/ST_SMCEX260SEC3_32Bit
TYPE ST_SMCEX260SEC3_32Bit :
STRUCT
	stOut AT %Q*: ST_SMCEX260SEC3_32Bit_Outputs;
END_STRUCT
END_TYPE

// SMC/ST_SMCEX260SEC3_32Bit_Outputs
TYPE ST_SMCEX260SEC3_32Bit_Outputs :
STRUCT
	bitOutput00: BIT;
	bitOutput01: BIT;
	bitOutput02: BIT;
	bitOutput03: BIT;
	bitOutput04: BIT;
	bitOutput05: BIT;
	bitOutput06: BIT;
	bitOutput07: BIT;
	
	bitOutput10: BIT;
	bitOutput11: BIT;
	bitOutput12: BIT;
	bitOutput13: BIT;
	bitOutput14: BIT;
	bitOutput15: BIT;
	bitOutput16: BIT;
	bitOutput17: BIT;
	
	bitOutput20: BIT;
	bitOutput21: BIT;
	bitOutput22: BIT;
	bitOutput23: BIT;
	bitOutput24: BIT;
	bitOutput25: BIT;
	bitOutput26: BIT;
	bitOutput27: BIT;
	
	bitOutput30: BIT;
	bitOutput31: BIT;
	bitOutput32: BIT;
	bitOutput33: BIT;
	bitOutput34: BIT;
	bitOutput35: BIT;
	bitOutput36: BIT;
	bitOutput37: BIT;

END_STRUCT
END_TYPE

// SMC/ST_SMCEX260SEC3_Outputs
TYPE ST_SMCEX260SEC3_Outputs :
STRUCT
	bitOutput00: BIT;
	bitOutput01: BIT;
	bitOutput02: BIT;
	bitOutput03: BIT;
	bitOutput04: BIT;
	bitOutput05: BIT;
	bitOutput06: BIT;
	bitOutput07: BIT;
	
	bitOutput10: BIT;
	bitOutput11: BIT;
	bitOutput12: BIT;
	bitOutput13: BIT;
	bitOutput14: BIT;
	bitOutput15: BIT;
	bitOutput16: BIT;
	bitOutput17: BIT;
END_STRUCT
END_TYPE

// IO Debug/F_LinkDigitalIOStructs
FUNCTION F_LinkDigitalIOStructs : BOOL
VAR_INPUT
END_VAR
VAR_IN_OUT
	(* The force and force value bits of this will be set to the values of the other. *)
	inout_stControl: ST_DebugDigitalIO;
	(* All info bits of this will be assigned to the control. *)
	inout_stStatus: ST_DebugDigitalIO;
END_VAR
VAR
END_VAR

inout_stStatus.bForce := inout_stControl.bForce;
inout_stStatus.bForceValue := inout_stControl.bForceValue;
inout_stControl.bCurrentValue := inout_stStatus.bCurrentValue;
inout_stControl.strLabel := inout_stStatus.strLabel;
inout_stControl.bOutput := inout_stStatus.bOutput;

END_FUNCTION

// IO Debug/F_SetDigitalInput
FUNCTION F_SetDigitalInput : BOOL
VAR_INPUT
	in_bValue: BOOL;
	in_strLabel: T_MaxString;
END_VAR
VAR_IN_OUT
	inout_stInput: ST_DebugDigitalIO;
END_VAR
VAR
END_VAR

inout_stInput.bOutput := FALSE;
inout_stInput.bCurrentValue := in_bValue;
inout_stInput.strLabel := in_strLabel;

END_FUNCTION

// IO Debug/F_SetDigitalOutput
FUNCTION F_SetDigitalOutput : BOOL
VAR_INPUT
	in_bValue: BOOL;
	in_strLabel: T_MaxString;
END_VAR
VAR_IN_OUT
	inout_stOutput: ST_DebugDigitalIO;
END_VAR
VAR_OUTPUT
	out_bValue: BOOL;
END_VAR
VAR
END_VAR

inout_stOutput.bOutput := TRUE;
inout_stOutput.strLabel := in_strLabel;
IF inout_stOutput.bForce THEN
	out_bValue := inout_stOutput.bForceValue;
ELSE
	out_bValue := in_bValue;
END_IF
inout_stOutput.bCurrentValue := out_bValue;

END_FUNCTION
